(* Logix 5000 project; controller Google vendor 1 type 14 code 151 rev 31.11; software revision 31.00; part 3 of 5 *)
(* tags used below, declared in another part *)
   API_AcceptFromAgv : BOOL;
   API_ScanRequest : BOOL;
   API_ScanRequestFWDTimer : TIMER;
   API_SendToAgv : BOOL;
   API_SendToAgvTimer : TIMER;
   Elev_FWD_Delay : TIMER;
   Elev_REV_Delay : TIMER;
   Elev_Slow : BOOL;
   FaultResetDelay : TIMER;
   HMI_AutoMode : BOOL;
   HMI_LiftJogDown : BOOL;
   HMI_LiftJogUp : BOOL;
   HMI_PB_Reset : BOOL;
   Infeed_Active : BOOL;
   Infeed_Upstream_ProdCode : DINT;
   Infeed_Upstream_ProdName : STRING;
   Infeed_Zone1 : Zone_Data;
   Infeed_Zone1_2_ProdCode : DINT;
   Infeed_Zone1_2_ProdName : STRING;
   Infeed_Zone1_FWD : BOOL;
   Infeed_Zone1_PE : BOOL;
   Infeed_Zone1_ProdCode : DINT;
   Infeed_Zone1_ProdName : STRING;
   Infeed_Zone1_REV : BOOL;
   Infeed_Zone2 : Zone_Data;
   Infeed_Zone2_3_ProdCode : DINT;
   Infeed_Zone2_3_ProdName : STRING;
   Infeed_Zone2_FWD : BOOL;
   Infeed_Zone2_PE : BOOL;
   Infeed_Zone2_ProdCode : DINT;
   Infeed_Zone2_ProdName : STRING;
   Infeed_Zone2_REV : BOOL;
   Infeed_Zone3 : Zone_Data;
   Infeed_Zone3_4_ProdCode : DINT;
   Infeed_Zone3_4_ProdName : STRING;
   Infeed_Zone3_FWD : BOOL;
   Infeed_Zone3_PE : BOOL;
   Infeed_Zone3_ProdCode : DINT;
   Infeed_Zone3_ProdName : STRING;
   Infeed_Zone3_REV : BOOL;
   Infeed_Zone4 : Zone_Data;
   Infeed_Zone4_FWD : BOOL;
   Infeed_Zone4_PE : BOOL;
   Infeed_Zone4_ProdCode : DINT;
   Infeed_Zone4_ProdName : STRING;
   Infeed_Zone4_REV : BOOL;
   Infeed_Zone_Timeout : TIMER[8];
   L1_CearOutResetTimer : TIMER;
   L1_Clear_Out : BOOL;
   L1_Zone1_FWD : BOOL;
   L1_Zone1_PE : BOOL;
   L2_Outfeed : BOOL;
   L2_Single_Outfeed : BOOL;
   L2_Z1_Outfeed : BOOL;
   L2_Z2_Outfeed : BOOL;
   L2_Z3_Outfeed : BOOL;
   L2_Z4_Outfeed : BOOL;
   L2_Zone1 : Zone_Data;
   L2_Zone2 : Zone_Data;
   L2_Zone3 : Zone_Data;
   L3_Outfeed : BOOL;
   L3_Single_Outfeed : BOOL;
   L3_Z1_Outfeed : BOOL;
   L3_Z2_Outfeed : BOOL;
   L3_Z3_Outfeed : BOOL;
   L3_Z4_Outfeed : BOOL;
   L3_Zone1 : Zone_Data;
   L3_Zone2 : Zone_Data;
   L3_Zone3 : Zone_Data;
   L4_Outfeed : BOOL;
   L4_Single_Outfeed : BOOL;
   L4_Z1_Outfeed : BOOL;
   L4_Z2_Outfeed : BOOL;
   L4_Z3_Outfeed : BOOL;
   L4_Z4_Outfeed : BOOL;
   L4_Zone1 : Zone_Data;
   L4_Zone2 : Zone_Data;
   L4_Zone3 : Zone_Data;
   L5_Outfeed : BOOL;
   L5_Single_Outfeed : BOOL;
   L5_Z1_Outfeed : BOOL;
   L5_Z2_Outfeed : BOOL;
   L5_Z3_Outfeed : BOOL;
   L5_Z4_Outfeed : BOOL;
   L5_Zone1 : Zone_Data;
   L5_Zone2 : Zone_Data;
   L5_Zone3 : Zone_Data;
   Level_1_Empty : BOOL;
   Level_2_Empty : BOOL;
   Level_2_Full : BOOL;
   Level_3_Empty : BOOL;
   Level_3_Full : BOOL;
   Level_4_Empty : BOOL;
   Level_4_Full : BOOL;
   Level_5_Empty : BOOL;
   Level_5_Full : BOOL;
   Lift_Alarm : BOOL;
   Lift_Ascend : BOOL;
   Lift_Current_Level : DINT;
   Lift_Cycle_Counter : COUNTER;
   Lift_Descend : BOOL;
   Lift_FullSpeed : DINT;
   Lift_L1_Slow_Prox : BOOL;
   Lift_L1_Stop_Prox : BOOL;
   Lift_L2_Slow_Prox : BOOL;
   Lift_L2_Stop_Prox : BOOL;
   Lift_L3_Slow_Prox : BOOL;
   Lift_L3_Stop_Prox : BOOL;
   Lift_L4_Slow_Prox : BOOL;
   Lift_L4_Stop_Prox : BOOL;
   Lift_L5_Slow_Prox : BOOL;
   Lift_L5_Stop_Prox : BOOL;
   Lift_Required_Level : DINT;
   Lift_SlowSpeed : DINT;
   Lift_Zone : Lift_Zone_Data;
   LiftZone_FWD : BOOL;
   LiftZone_REV : BOOL;
   LiftZoneDownstream_ProdCode : DINT;
   LiftZoneUpstream_ProdName : STRING;
   Motion_Complete : BOOL;
   ONS : DINT[6];
   Outfeed_Active : BOOL;
   Outfeed_Automatic : BOOL;
   Outfeed_Batch : BOOL;
   Outfeed_Single : BOOL;
   Safety_Relay_Status : BOOL;
   Sort_Number : DINT;
   Sorting_Active : BOOL;
   Sorting_Inactive : BOOL;
   System : State;
   System_Mode_Change : BOOL;
   System_State : DINT;
(* MainProgram, continued *)

ROUTINE R04_Sorting   (* ladder *)
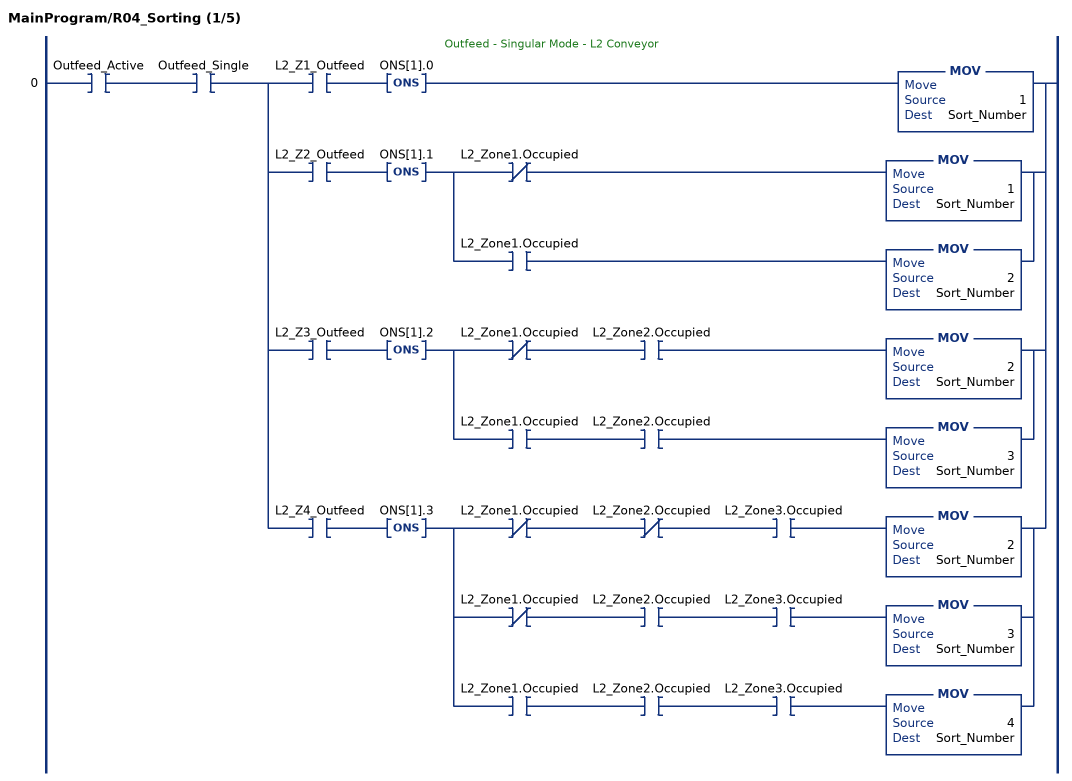
   // Outfeed - Singular Mode - L2 Conveyor
   0: XIC(Outfeed_Active)XIC(Outfeed_Single)[XIC(L2_Z1_Outfeed) ONS(ONS[1].0) MOV(1,Sort_Number) ,XIC(L2_Z2_Outfeed) ONS(ONS[1].1) [XIO(L2_Zone1.Occupied) MOV(1,Sort_Number) ,XIC(L2_Zone1.Occupied) MOV(2,Sort_Number) ] ,XIC(L2_Z3_Outfeed) ONS(ONS[1].2) [XIO(L2_Zone1.Occupied) XIC(L2_Zone2.Occupied) MOV(2,Sort_Number) ,XIC(L2_Zone1.Occupied) XIC(L2_Zone2.Occupied) MOV(3,Sort_Number) ] ,XIC(L2_Z4_Outfeed) ONS(ONS[1].3) [XIO(L2_Zone1.Occupied) XIO(L2_Zone2.Occupied) XIC(L2_Zone3.Occupied) MOV(2,Sort_Number) ,XIO(L2_Zone1.Occupied) XIC(L2_Zone2.Occupied) XIC(L2_Zone3.Occupied) MOV(3,Sort_Number) ,XIC(L2_Zone1.Occupied) XIC(L2_Zone2.Occupied) XIC(L2_Zone3.Occupied) MOV(4,Sort_Number) ] ];
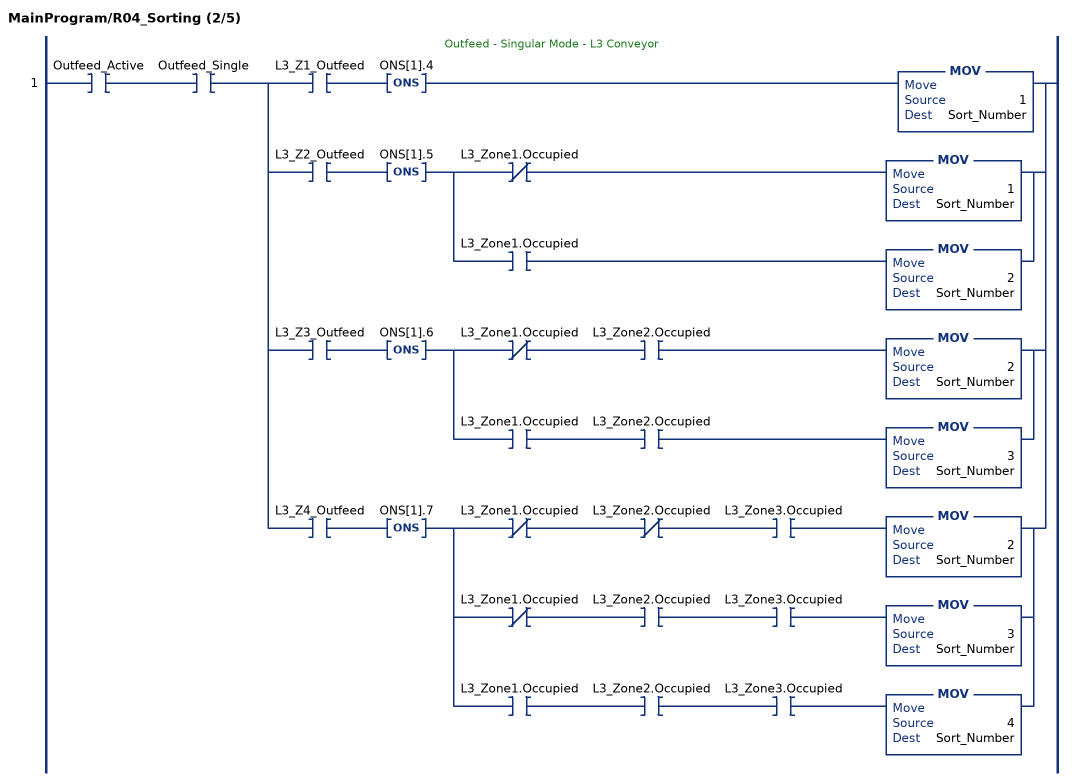
   // Outfeed - Singular Mode - L3 Conveyor
   1: XIC(Outfeed_Active)XIC(Outfeed_Single)[XIC(L3_Z1_Outfeed) ONS(ONS[1].4) MOV(1,Sort_Number) ,XIC(L3_Z2_Outfeed) ONS(ONS[1].5) [XIO(L3_Zone1.Occupied) MOV(1,Sort_Number) ,XIC(L3_Zone1.Occupied) MOV(2,Sort_Number) ] ,XIC(L3_Z3_Outfeed) ONS(ONS[1].6) [XIO(L3_Zone1.Occupied) XIC(L3_Zone2.Occupied) MOV(2,Sort_Number) ,XIC(L3_Zone1.Occupied) XIC(L3_Zone2.Occupied) MOV(3,Sort_Number) ] ,XIC(L3_Z4_Outfeed) ONS(ONS[1].7) [XIO(L3_Zone1.Occupied) XIO(L3_Zone2.Occupied) XIC(L3_Zone3.Occupied) MOV(2,Sort_Number) ,XIO(L3_Zone1.Occupied) XIC(L3_Zone2.Occupied) XIC(L3_Zone3.Occupied) MOV(3,Sort_Number) ,XIC(L3_Zone1.Occupied) XIC(L3_Zone2.Occupied) XIC(L3_Zone3.Occupied) MOV(4,Sort_Number) ] ];
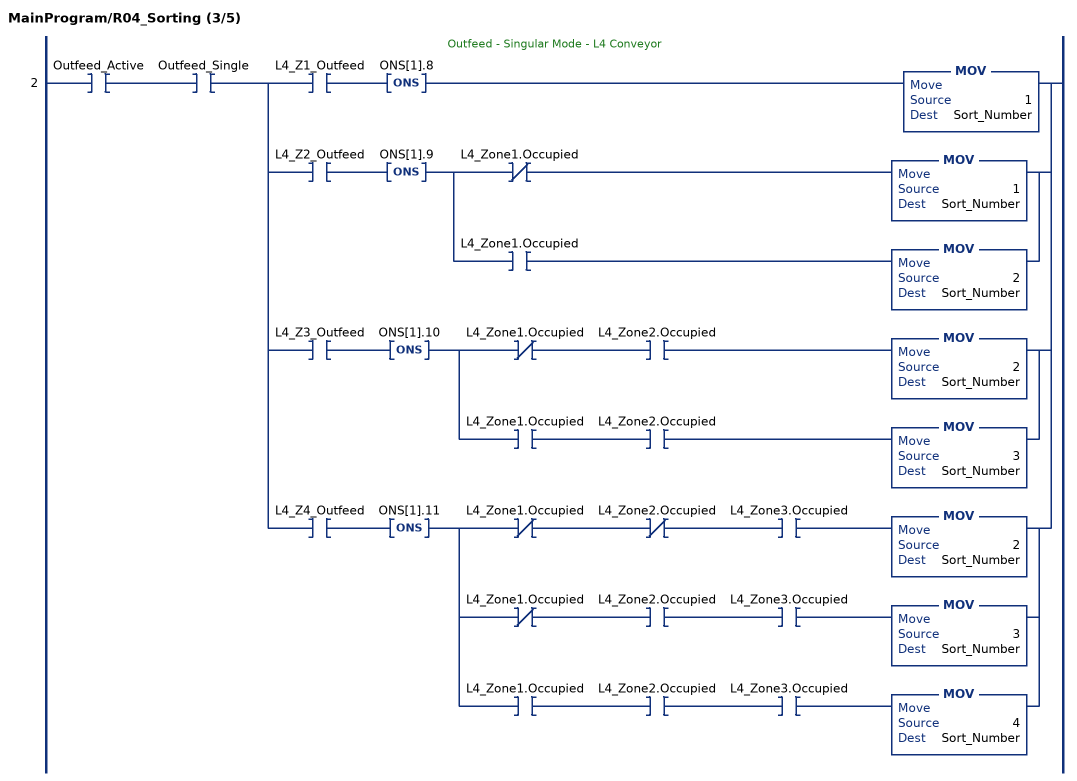
   // Outfeed - Singular Mode - L4 Conveyor
   2: XIC(Outfeed_Active)XIC(Outfeed_Single)[XIC(L4_Z1_Outfeed) ONS(ONS[1].8) MOV(1,Sort_Number) ,XIC(L4_Z2_Outfeed) ONS(ONS[1].9) [XIO(L4_Zone1.Occupied) MOV(1,Sort_Number) ,XIC(L4_Zone1.Occupied) MOV(2,Sort_Number) ] ,XIC(L4_Z3_Outfeed) ONS(ONS[1].10) [XIO(L4_Zone1.Occupied) XIC(L4_Zone2.Occupied) MOV(2,Sort_Number) ,XIC(L4_Zone1.Occupied) XIC(L4_Zone2.Occupied) MOV(3,Sort_Number) ] ,XIC(L4_Z4_Outfeed) ONS(ONS[1].11) [XIO(L4_Zone1.Occupied) XIO(L4_Zone2.Occupied) XIC(L4_Zone3.Occupied) MOV(2,Sort_Number) ,XIO(L4_Zone1.Occupied) XIC(L4_Zone2.Occupied) XIC(L4_Zone3.Occupied) MOV(3,Sort_Number) ,XIC(L4_Zone1.Occupied) XIC(L4_Zone2.Occupied) XIC(L4_Zone3.Occupied) MOV(4,Sort_Number) ] ];
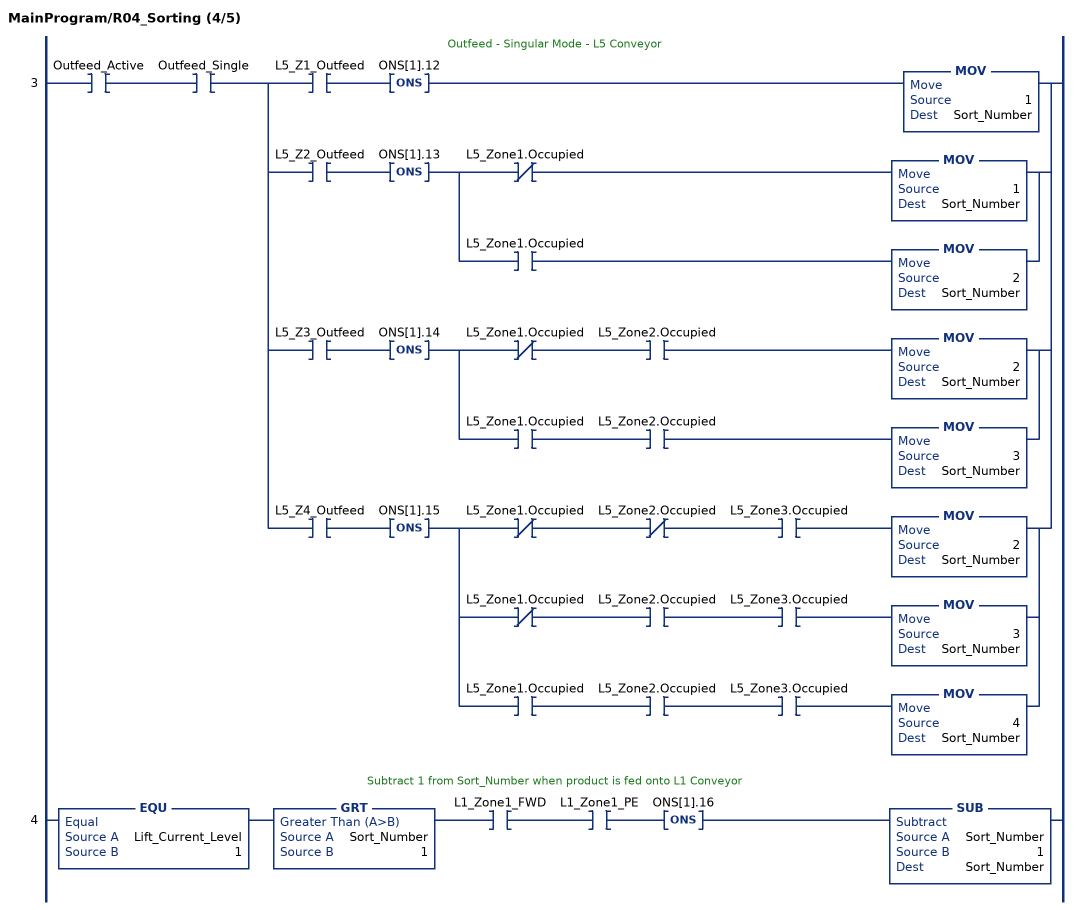
   // Outfeed - Singular Mode - L5 Conveyor
   3: XIC(Outfeed_Active)XIC(Outfeed_Single)[XIC(L5_Z1_Outfeed) ONS(ONS[1].12) MOV(1,Sort_Number) ,XIC(L5_Z2_Outfeed) ONS(ONS[1].13) [XIO(L5_Zone1.Occupied) MOV(1,Sort_Number) ,XIC(L5_Zone1.Occupied) MOV(2,Sort_Number) ] ,XIC(L5_Z3_Outfeed) ONS(ONS[1].14) [XIO(L5_Zone1.Occupied) XIC(L5_Zone2.Occupied) MOV(2,Sort_Number) ,XIC(L5_Zone1.Occupied) XIC(L5_Zone2.Occupied) MOV(3,Sort_Number) ] ,XIC(L5_Z4_Outfeed) ONS(ONS[1].15) [XIO(L5_Zone1.Occupied) XIO(L5_Zone2.Occupied) XIC(L5_Zone3.Occupied) MOV(2,Sort_Number) ,XIO(L5_Zone1.Occupied) XIC(L5_Zone2.Occupied) XIC(L5_Zone3.Occupied) MOV(3,Sort_Number) ,XIC(L5_Zone1.Occupied) XIC(L5_Zone2.Occupied) XIC(L5_Zone3.Occupied) MOV(4,Sort_Number) ] ];
   // Subtract 1 from Sort_Number when product is fed onto L1 Conveyor
   4: EQU(Lift_Current_Level,1)GRT(Sort_Number,1)XIC(L1_Zone1_FWD)XIC(L1_Zone1_PE)ONS(ONS[1].16)SUB(Sort_Number,1,Sort_Number);
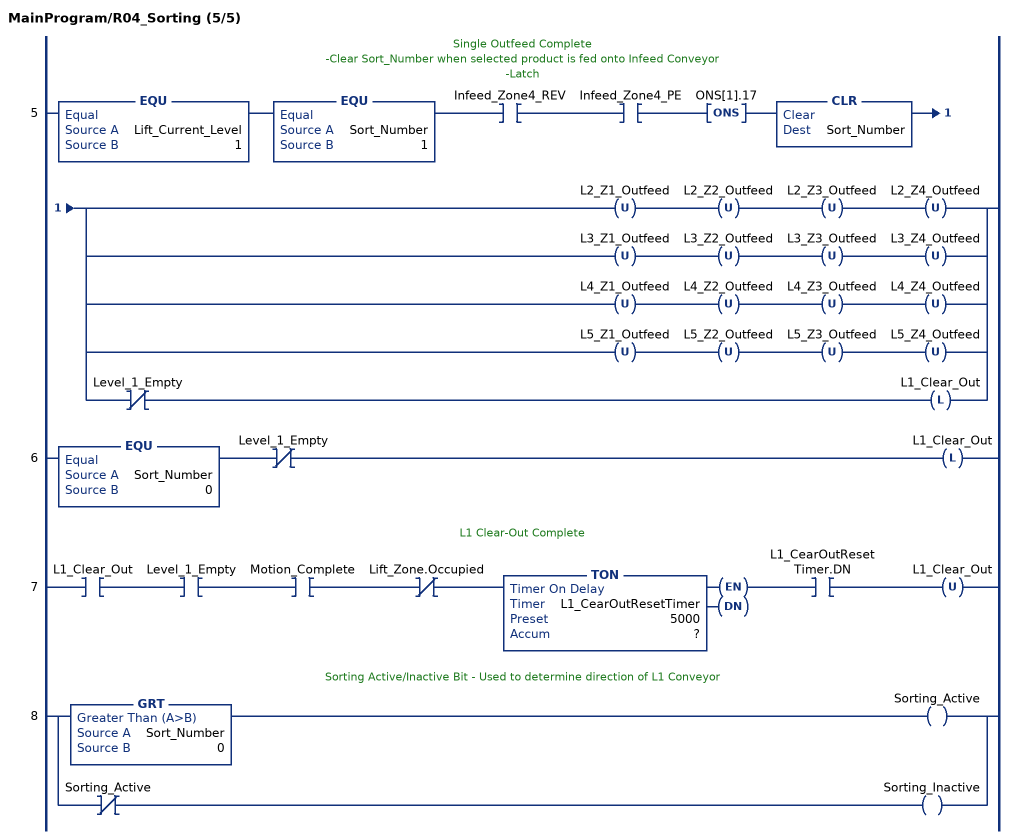
   // Single Outfeed Complete
   // -Clear Sort_Number when selected product is fed onto Infeed Conveyor
   // -Latch
   5: EQU(Lift_Current_Level,1)EQU(Sort_Number,1)XIC(Infeed_Zone4_REV)XIC(Infeed_Zone4_PE)ONS(ONS[1].17)CLR(Sort_Number)[OTU(L2_Z1_Outfeed) OTU(L2_Z2_Outfeed) OTU(L2_Z3_Outfeed) OTU(L2_Z4_Outfeed) ,OTU(L3_Z1_Outfeed) OTU(L3_Z2_Outfeed) OTU(L3_Z3_Outfeed) OTU(L3_Z4_Outfeed) ,OTU(L4_Z1_Outfeed) OTU(L4_Z2_Outfeed) OTU(L4_Z3_Outfeed) OTU(L4_Z4_Outfeed) ,OTU(L5_Z1_Outfeed) OTU(L5_Z2_Outfeed) OTU(L5_Z3_Outfeed) OTU(L5_Z4_Outfeed) ,XIO(Level_1_Empty) OTL(L1_Clear_Out) ];
   6: EQU(Sort_Number,0)XIO(Level_1_Empty)OTL(L1_Clear_Out);
   // L1 Clear-Out Complete
   7: XIC(L1_Clear_Out)XIC(Level_1_Empty)XIC(Motion_Complete)XIO(Lift_Zone.Occupied)TON(L1_CearOutResetTimer,?,?)XIC(L1_CearOutResetTimer.DN)OTU(L1_Clear_Out);
   // Sorting Active/Inactive Bit - Used to determine direction of L1 Conveyor
   8: [GRT(Sort_Number,0) OTE(Sorting_Active) ,XIO(Sorting_Active) OTE(Sorting_Inactive) ];
END_ROUTINE

ROUTINE R05_Lift_Level_Selection   (* ladder *)
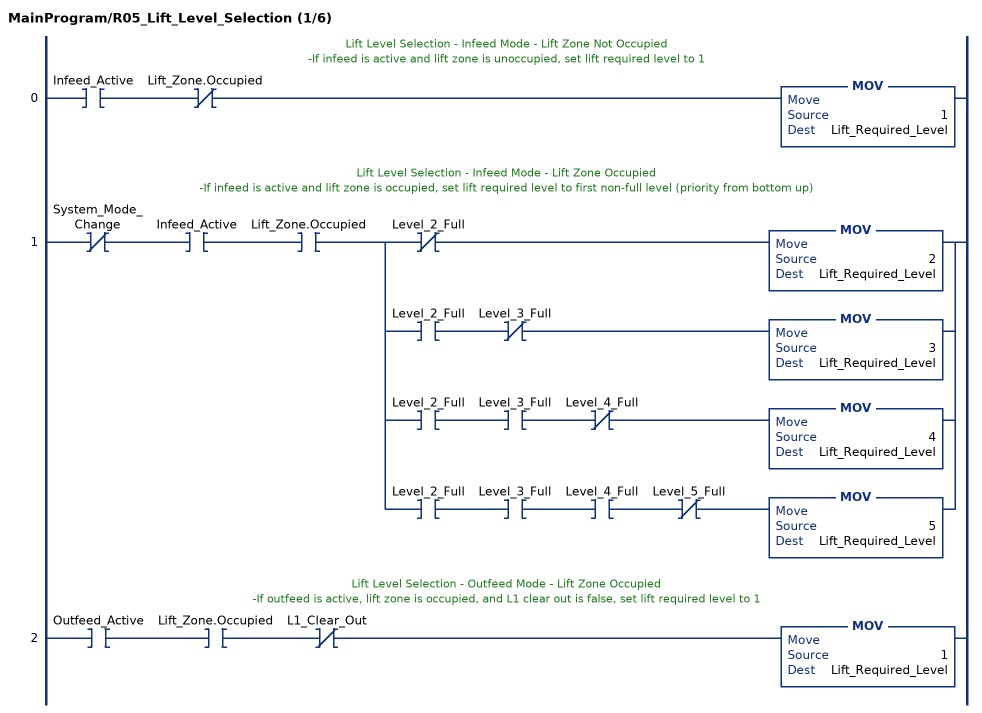
   // Lift Level Selection - Infeed Mode - Lift Zone Not Occupied
   // -If infeed is active and lift zone is unoccupied, set lift required level to 1
   0: XIC(Infeed_Active)XIO(Lift_Zone.Occupied)MOV(1,Lift_Required_Level);
   // Lift Level Selection - Infeed Mode - Lift Zone Occupied
   // -If infeed is active and lift zone is occupied, set lift required level to first non-full level (priority from bottom up)
   1: XIO(System_Mode_Change)XIC(Infeed_Active)XIC(Lift_Zone.Occupied)[XIO(Level_2_Full) MOV(2,Lift_Required_Level) ,XIC(Level_2_Full) XIO(Level_3_Full) MOV(3,Lift_Required_Level) ,XIC(Level_2_Full) XIC(Level_3_Full) XIO(Level_4_Full) MOV(4,Lift_Required_Level) ,XIC(Level_2_Full) XIC(Level_3_Full) XIC(Level_4_Full) XIO(Level_5_Full) MOV(5,Lift_Required_Level) ];
   // Lift Level Selection - Outfeed Mode - Lift Zone Occupied
   // -If outfeed is active, lift zone is occupied, and L1 clear out is false, set lift required level to 1
   2: XIC(Outfeed_Active)XIC(Lift_Zone.Occupied)XIO(L1_Clear_Out)MOV(1,Lift_Required_Level);
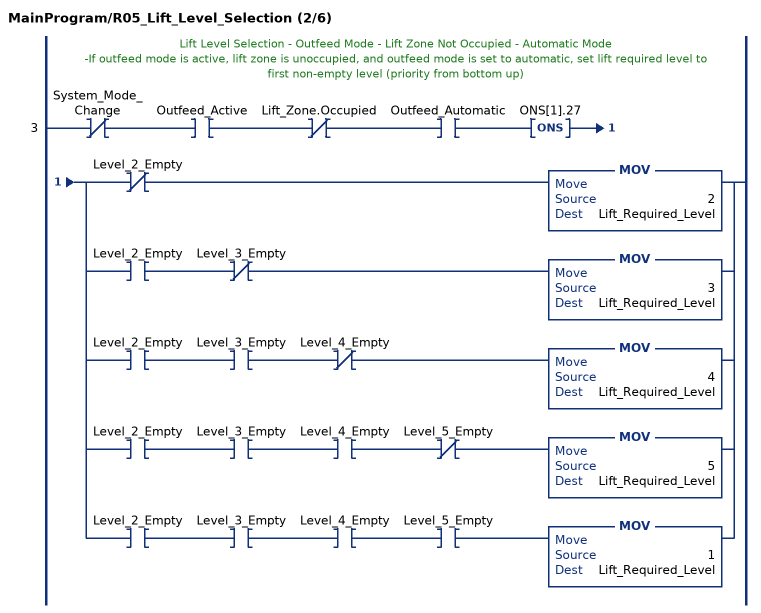
   // Lift Level Selection - Outfeed Mode - Lift Zone Not Occupied - Automatic Mode
   // -If outfeed mode is active, lift zone is unoccupied, and outfeed mode is set to automatic, set lift required level to first non-empty level (priority from bottom up)
   3: XIO(System_Mode_Change)XIC(Outfeed_Active)XIO(Lift_Zone.Occupied)XIC(Outfeed_Automatic)ONS(ONS[1].27)[XIO(Level_2_Empty) MOV(2,Lift_Required_Level) ,XIC(Level_2_Empty) XIO(Level_3_Empty) MOV(3,Lift_Required_Level) ,XIC(Level_2_Empty) XIC(Level_3_Empty) XIO(Level_4_Empty) MOV(4,Lift_Required_Level) ,XIC(Level_2_Empty) XIC(Level_3_Empty) XIC(Level_4_Empty) XIO(Level_5_Empty) MOV(5,Lift_Required_Level) ,XIC(Level_2_Empty) XIC(Level_3_Empty) XIC(Level_4_Empty) XIC(Level_5_Empty) MOV(1,Lift_Required_Level) ];
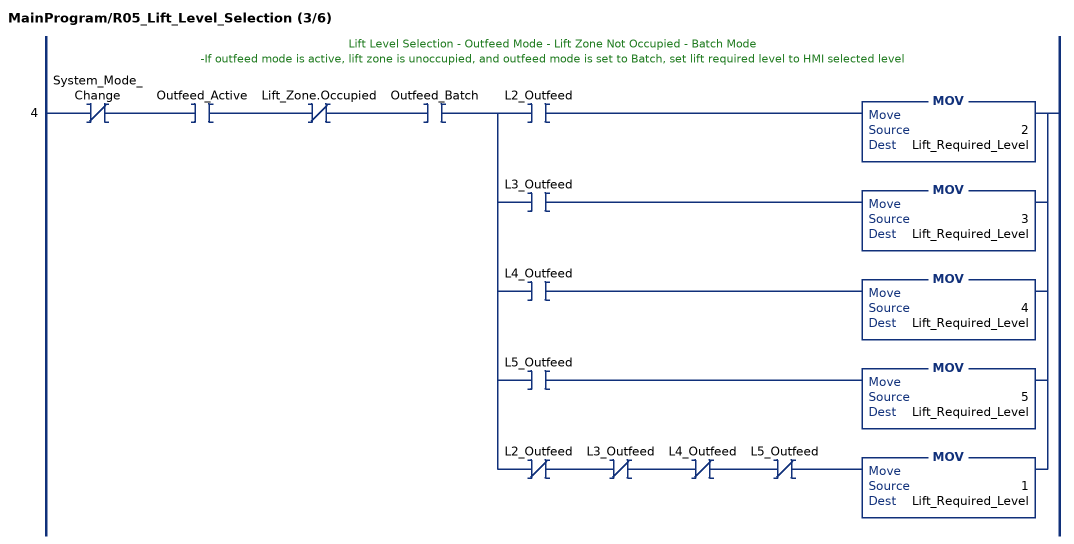
   // Lift Level Selection - Outfeed Mode - Lift Zone Not Occupied - Batch Mode
   // -If outfeed mode is active, lift zone is unoccupied, and outfeed mode is set to Batch, set lift required level to HMI selected level
   4: XIO(System_Mode_Change)XIC(Outfeed_Active)XIO(Lift_Zone.Occupied)XIC(Outfeed_Batch)[XIC(L2_Outfeed) MOV(2,Lift_Required_Level) ,XIC(L3_Outfeed) MOV(3,Lift_Required_Level) ,XIC(L4_Outfeed) MOV(4,Lift_Required_Level) ,XIC(L5_Outfeed) MOV(5,Lift_Required_Level) ,XIO(L2_Outfeed) XIO(L3_Outfeed) XIO(L4_Outfeed) XIO(L5_Outfeed) MOV(1,Lift_Required_Level) ];
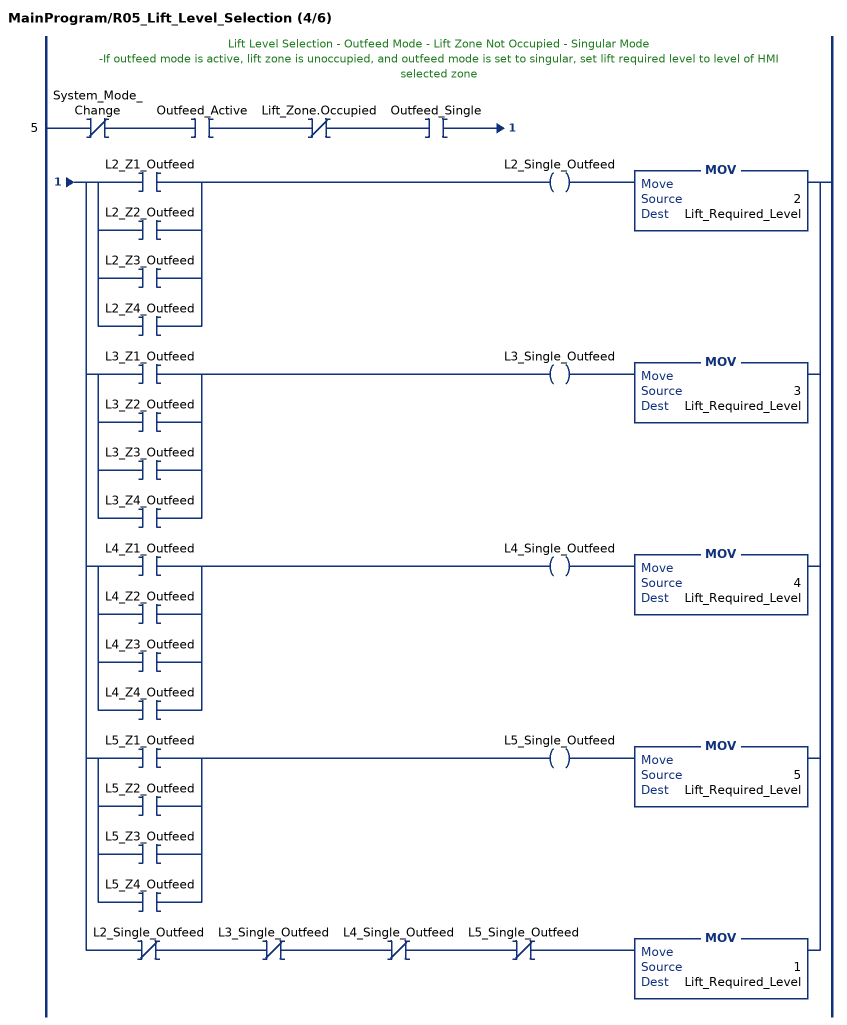
   // Lift Level Selection - Outfeed Mode - Lift Zone Not Occupied - Singular Mode
   // -If outfeed mode is active, lift zone is unoccupied, and outfeed mode is set to singular, set lift required level to level of HMI selected zone
   5: XIO(System_Mode_Change)XIC(Outfeed_Active)XIO(Lift_Zone.Occupied)XIC(Outfeed_Single)[[XIC(L2_Z1_Outfeed) ,XIC(L2_Z2_Outfeed) ,XIC(L2_Z3_Outfeed) ,XIC(L2_Z4_Outfeed) ] OTE(L2_Single_Outfeed) MOV(2,Lift_Required_Level) ,[XIC(L3_Z1_Outfeed) ,XIC(L3_Z2_Outfeed) ,XIC(L3_Z3_Outfeed) ,XIC(L3_Z4_Outfeed) ] OTE(L3_Single_Outfeed) MOV(3,Lift_Required_Level) ,[XIC(L4_Z1_Outfeed) ,XIC(L4_Z2_Outfeed) ,XIC(L4_Z3_Outfeed) ,XIC(L4_Z4_Outfeed) ] OTE(L4_Single_Outfeed) MOV(4,Lift_Required_Level) ,[XIC(L5_Z1_Outfeed) ,XIC(L5_Z2_Outfeed) ,XIC(L5_Z3_Outfeed) ,XIC(L5_Z4_Outfeed) ] OTE(L5_Single_Outfeed) MOV(5,Lift_Required_Level) ,XIO(L2_Single_Outfeed) XIO(L3_Single_Outfeed) XIO(L4_Single_Outfeed) XIO(L5_Single_Outfeed) MOV(1,Lift_Required_Level) ];
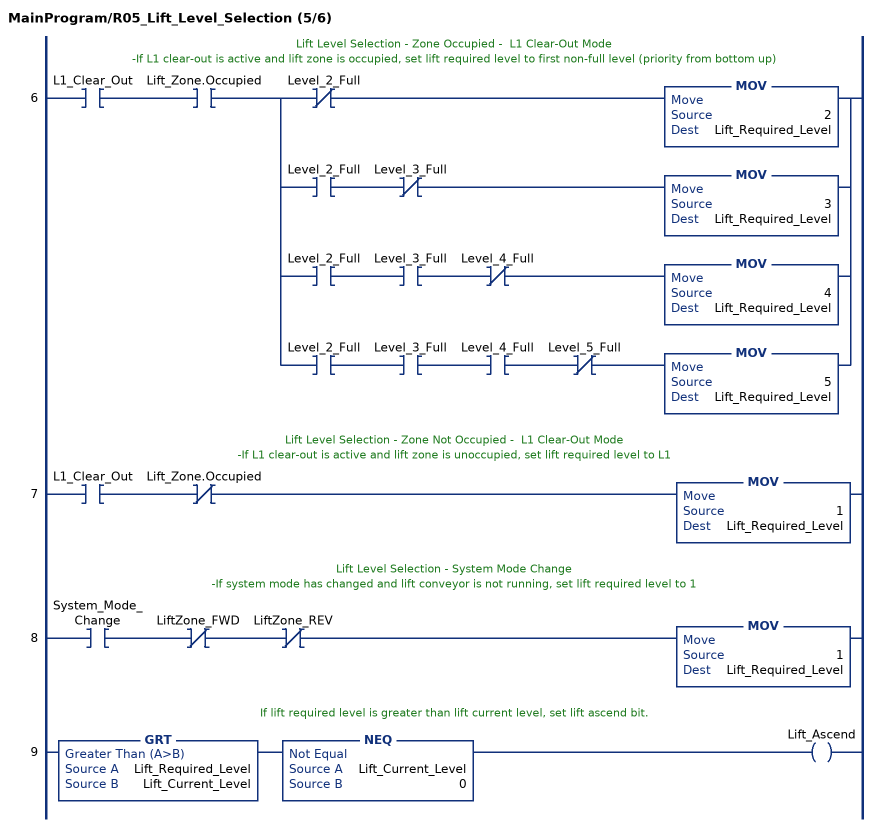
   // Lift Level Selection - Zone Occupied -  L1 Clear-Out Mode
   // -If L1 clear-out is active and lift zone is occupied, set lift required level to first non-full level (priority from bottom up)
   6: XIC(L1_Clear_Out)XIC(Lift_Zone.Occupied)[XIO(Level_2_Full) MOV(2,Lift_Required_Level) ,XIC(Level_2_Full) XIO(Level_3_Full) MOV(3,Lift_Required_Level) ,XIC(Level_2_Full) XIC(Level_3_Full) XIO(Level_4_Full) MOV(4,Lift_Required_Level) ,XIC(Level_2_Full) XIC(Level_3_Full) XIC(Level_4_Full) XIO(Level_5_Full) MOV(5,Lift_Required_Level) ];
   // Lift Level Selection - Zone Not Occupied -  L1 Clear-Out Mode
   // -If L1 clear-out is active and lift zone is unoccupied, set lift required level to L1
   7: XIC(L1_Clear_Out)XIO(Lift_Zone.Occupied)MOV(1,Lift_Required_Level);
   // Lift Level Selection - System Mode Change
   // -If system mode has changed and lift conveyor is not running, set lift required level to 1
   8: XIC(System_Mode_Change)XIO(LiftZone_FWD)XIO(LiftZone_REV)MOV(1,Lift_Required_Level);
   // If lift required level is greater than lift current level, set lift ascend bit.
   9: GRT(Lift_Required_Level,Lift_Current_Level)NEQ(Lift_Current_Level,0)OTE(Lift_Ascend);
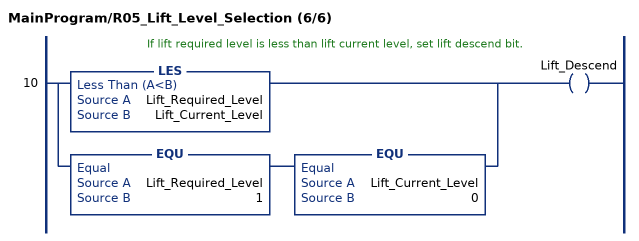
   // If lift required level is less than lift current level, set lift descend bit.
   10: [LES(Lift_Required_Level,Lift_Current_Level) ,EQU(Lift_Required_Level,1) EQU(Lift_Current_Level,0) ]OTE(Lift_Descend);
END_ROUTINE

ROUTINE R06_Lift_Operation   (* ladder *)
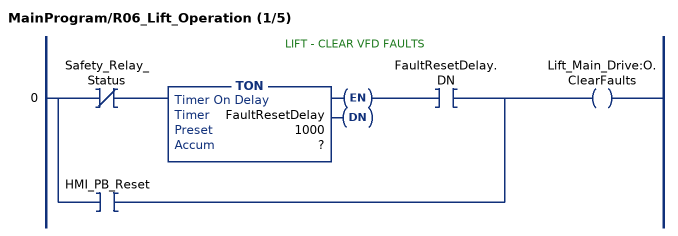
   // LIFT - CLEAR VFD FAULTS
   0: [XIO(Safety_Relay_Status) TON(FaultResetDelay,?,?) XIC(FaultResetDelay.DN) ,XIC(HMI_PB_Reset) ]OTE(Lift_Main_Drive:O.ClearFaults);
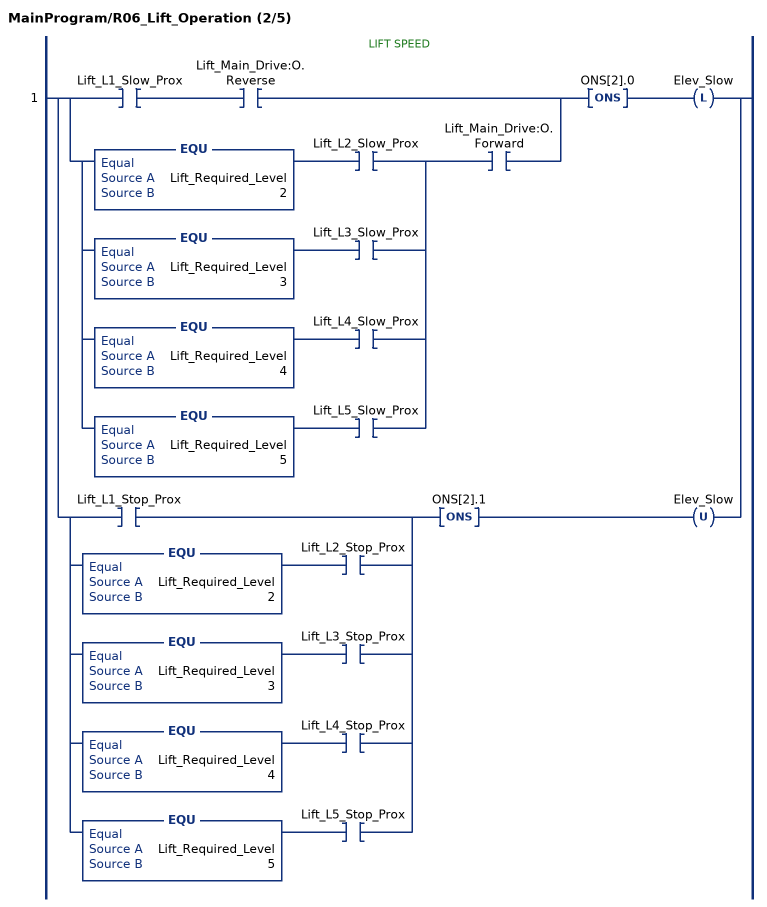
   // LIFT SPEED
   1: [[XIC(Lift_L1_Slow_Prox) XIC(Lift_Main_Drive:O.Reverse) ,[EQU(Lift_Required_Level,2) XIC(Lift_L2_Slow_Prox) ,EQU(Lift_Required_Level,3) XIC(Lift_L3_Slow_Prox) ,EQU(Lift_Required_Level,4) XIC(Lift_L4_Slow_Prox) ,EQU(Lift_Required_Level,5) XIC(Lift_L5_Slow_Prox) ] XIC(Lift_Main_Drive:O.Forward) ] ONS(ONS[2].0) OTL(Elev_Slow) ,[XIC(Lift_L1_Stop_Prox) ,EQU(Lift_Required_Level,2) XIC(Lift_L2_Stop_Prox) ,EQU(Lift_Required_Level,3) XIC(Lift_L3_Stop_Prox) ,EQU(Lift_Required_Level,4) XIC(Lift_L4_Stop_Prox) ,EQU(Lift_Required_Level,5) XIC(Lift_L5_Stop_Prox) ] ONS(ONS[2].1) OTU(Elev_Slow) ];
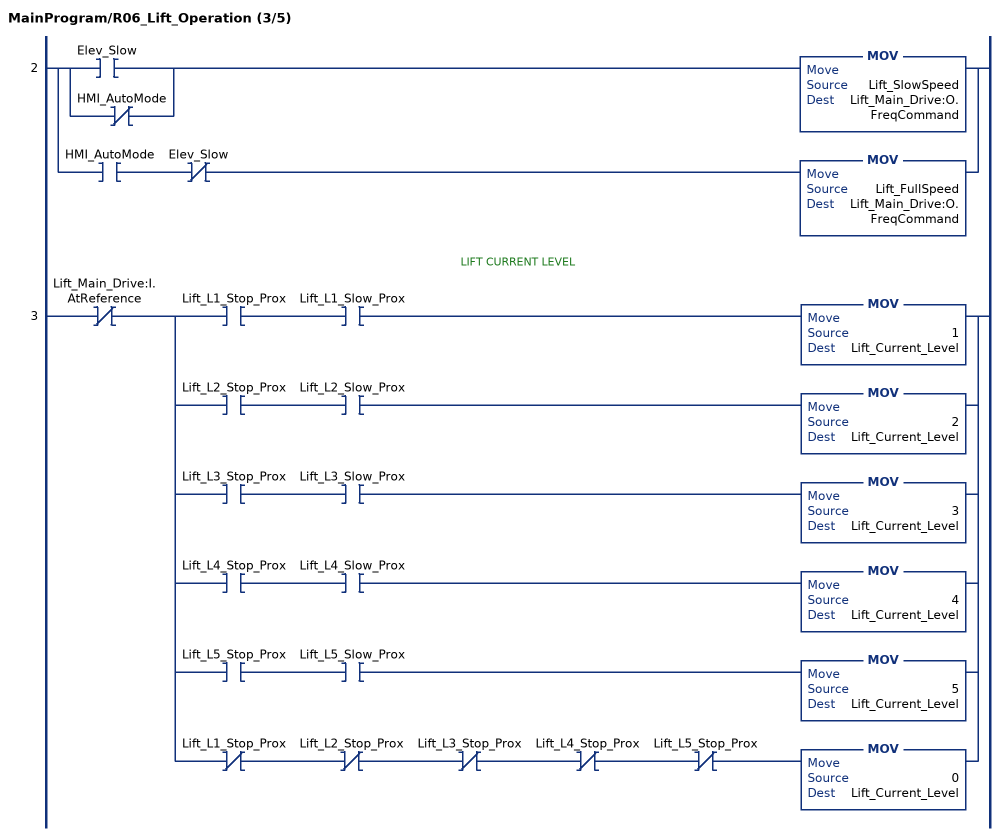
   2: [[XIC(Elev_Slow) ,XIO(HMI_AutoMode) ] MOV(Lift_SlowSpeed,Lift_Main_Drive:O.FreqCommand) ,XIC(HMI_AutoMode) XIO(Elev_Slow) MOV(Lift_FullSpeed,Lift_Main_Drive:O.FreqCommand) ];
   // LIFT CURRENT LEVEL
   3: XIO(Lift_Main_Drive:I.AtReference)[XIC(Lift_L1_Stop_Prox) XIC(Lift_L1_Slow_Prox) MOV(1,Lift_Current_Level) ,XIC(Lift_L2_Stop_Prox) XIC(Lift_L2_Slow_Prox) MOV(2,Lift_Current_Level) ,XIC(Lift_L3_Stop_Prox) XIC(Lift_L3_Slow_Prox) MOV(3,Lift_Current_Level) ,XIC(Lift_L4_Stop_Prox) XIC(Lift_L4_Slow_Prox) MOV(4,Lift_Current_Level) ,XIC(Lift_L5_Stop_Prox) XIC(Lift_L5_Slow_Prox) MOV(5,Lift_Current_Level) ,XIO(Lift_L1_Stop_Prox) XIO(Lift_L2_Stop_Prox) XIO(Lift_L3_Stop_Prox) XIO(Lift_L4_Stop_Prox) XIO(Lift_L5_Stop_Prox) MOV(0,Lift_Current_Level) ];
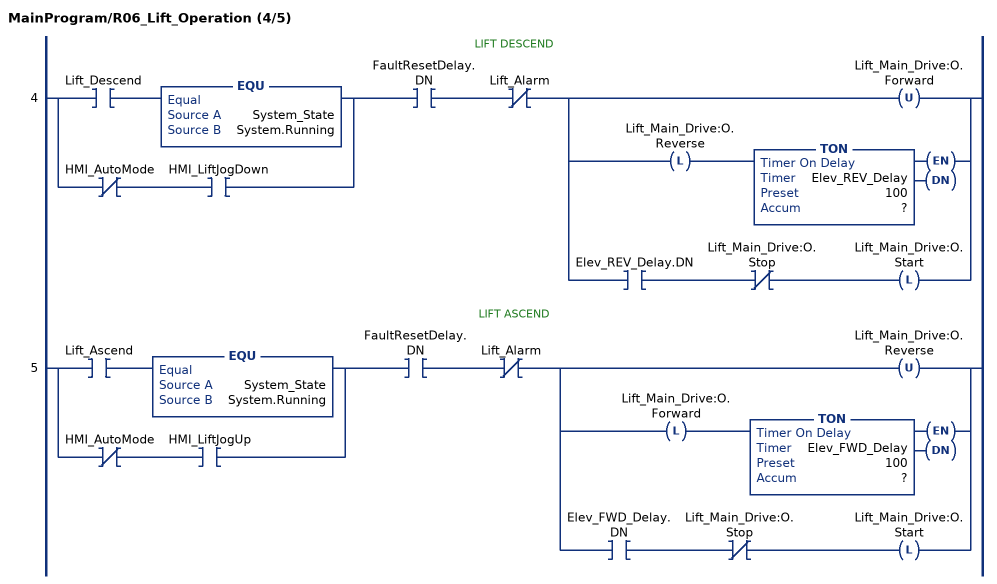
   // LIFT DESCEND
   4: [XIC(Lift_Descend) EQU(System_State,System.Running) ,XIO(HMI_AutoMode) XIC(HMI_LiftJogDown) ]XIC(FaultResetDelay.DN)XIO(Lift_Alarm)[OTU(Lift_Main_Drive:O.Forward) ,OTL(Lift_Main_Drive:O.Reverse) TON(Elev_REV_Delay,?,?) ,XIC(Elev_REV_Delay.DN) XIO(Lift_Main_Drive:O.Stop) OTL(Lift_Main_Drive:O.Start) ];
   // LIFT ASCEND
   5: [XIC(Lift_Ascend) EQU(System_State,System.Running) ,XIO(HMI_AutoMode) XIC(HMI_LiftJogUp) ]XIC(FaultResetDelay.DN)XIO(Lift_Alarm)[OTU(Lift_Main_Drive:O.Reverse) ,OTL(Lift_Main_Drive:O.Forward) TON(Elev_FWD_Delay,?,?) ,XIC(Elev_FWD_Delay.DN) XIO(Lift_Main_Drive:O.Stop) OTL(Lift_Main_Drive:O.Start) ];
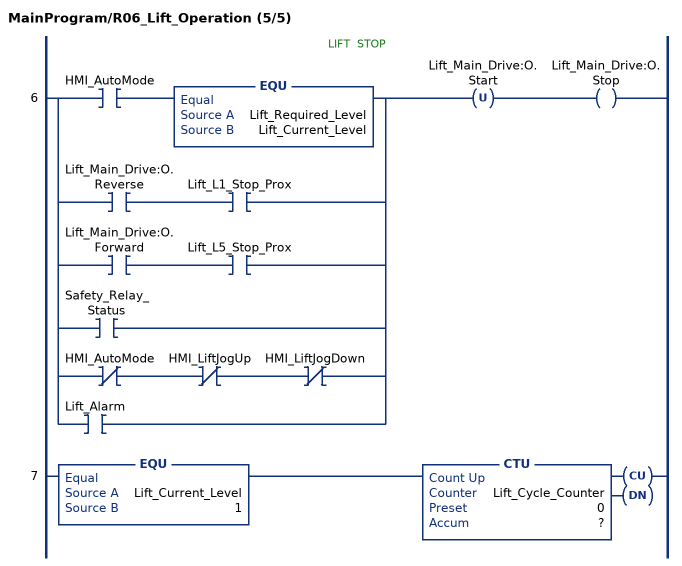
   // LIFT  STOP
   6: [XIC(HMI_AutoMode) EQU(Lift_Required_Level,Lift_Current_Level) ,XIC(Lift_Main_Drive:O.Reverse) XIC(Lift_L1_Stop_Prox) ,XIC(Lift_Main_Drive:O.Forward) XIC(Lift_L5_Stop_Prox) ,XIC(Safety_Relay_Status) ,XIO(HMI_AutoMode) XIO(HMI_LiftJogUp) XIO(HMI_LiftJogDown) ,XIC(Lift_Alarm) ]OTU(Lift_Main_Drive:O.Start)OTE(Lift_Main_Drive:O.Stop);
   7: EQU(Lift_Current_Level,1)CTU(Lift_Cycle_Counter,?,?);
END_ROUTINE

ROUTINE R07_Infeed_Conveyor   (* ladder *)
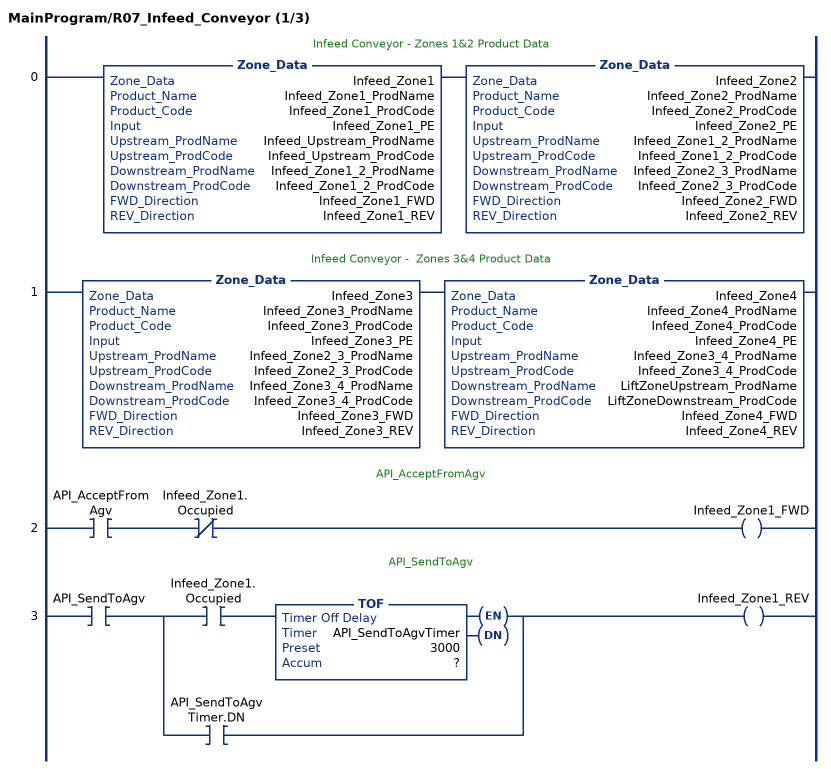
   // Infeed Conveyor - Zones 1&2 Product Data
   0: Zone_Data(Infeed_Zone1,Infeed_Zone1_ProdName,Infeed_Zone1_ProdCode,Infeed_Zone1_PE,Infeed_Upstream_ProdName,Infeed_Upstream_ProdCode,Infeed_Zone1_2_ProdName,Infeed_Zone1_2_ProdCode,Infeed_Zone1_FWD,Infeed_Zone1_REV)Zone_Data(Infeed_Zone2,Infeed_Zone2_ProdName,Infeed_Zone2_ProdCode,Infeed_Zone2_PE,Infeed_Zone1_2_ProdName,Infeed_Zone1_2_ProdCode,Infeed_Zone2_3_ProdName,Infeed_Zone2_3_ProdCode,Infeed_Zone2_FWD,Infeed_Zone2_REV);
   // Infeed Conveyor -  Zones 3&4 Product Data
   1: Zone_Data(Infeed_Zone3,Infeed_Zone3_ProdName,Infeed_Zone3_ProdCode,Infeed_Zone3_PE,Infeed_Zone2_3_ProdName,Infeed_Zone2_3_ProdCode,Infeed_Zone3_4_ProdName,Infeed_Zone3_4_ProdCode,Infeed_Zone3_FWD,Infeed_Zone3_REV)Zone_Data(Infeed_Zone4,Infeed_Zone4_ProdName,Infeed_Zone4_ProdCode,Infeed_Zone4_PE,Infeed_Zone3_4_ProdName,Infeed_Zone3_4_ProdCode,LiftZoneUpstream_ProdName,LiftZoneDownstream_ProdCode,Infeed_Zone4_FWD,Infeed_Zone4_REV);
   // API_AcceptFromAgv
   2: XIC(API_AcceptFromAgv)XIO(Infeed_Zone1.Occupied)OTE(Infeed_Zone1_FWD);
   // API_SendToAgv
   3: XIC(API_SendToAgv)[XIC(Infeed_Zone1.Occupied) TOF(API_SendToAgvTimer,?,?) ,XIC(API_SendToAgvTimer.DN) ]OTE(Infeed_Zone1_REV);
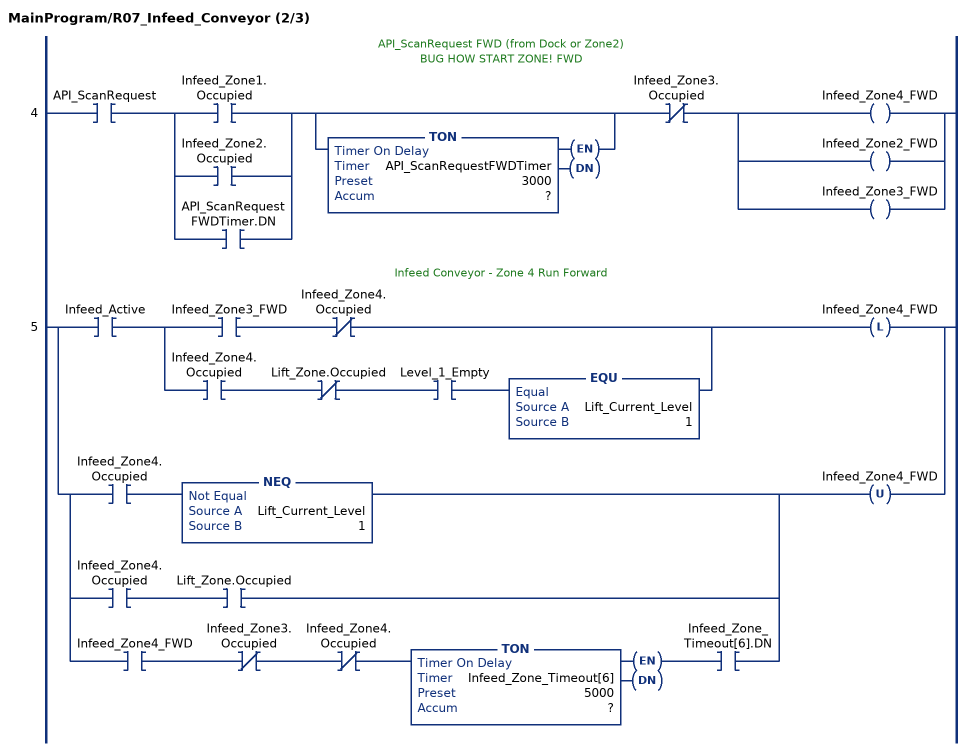
   // API_ScanRequest FWD (from Dock or Zone2)
   // BUG HOW START ZONE! FWD
   4: XIC(API_ScanRequest)[XIC(Infeed_Zone1.Occupied) ,XIC(Infeed_Zone2.Occupied) ,XIC(API_ScanRequestFWDTimer.DN) ][,TON(API_ScanRequestFWDTimer,?,?) ]XIO(Infeed_Zone3.Occupied)[OTE(Infeed_Zone4_FWD) ,OTE(Infeed_Zone2_FWD) ,OTE(Infeed_Zone3_FWD) ];
   // Infeed Conveyor - Zone 4 Run Forward
   5: [XIC(Infeed_Active) [XIC(Infeed_Zone3_FWD) XIO(Infeed_Zone4.Occupied) ,XIC(Infeed_Zone4.Occupied) XIO(Lift_Zone.Occupied) XIC(Level_1_Empty) EQU(Lift_Current_Level,1) ] OTL(Infeed_Zone4_FWD) ,[XIC(Infeed_Zone4.Occupied) NEQ(Lift_Current_Level,1) ,XIC(Infeed_Zone4.Occupied) XIC(Lift_Zone.Occupied) ,XIC(Infeed_Zone4_FWD) XIO(Infeed_Zone3.Occupied) XIO(Infeed_Zone4.Occupied) TON(Infeed_Zone_Timeout[6],?,?) XIC(Infeed_Zone_Timeout[6].DN) ] OTU(Infeed_Zone4_FWD) ];
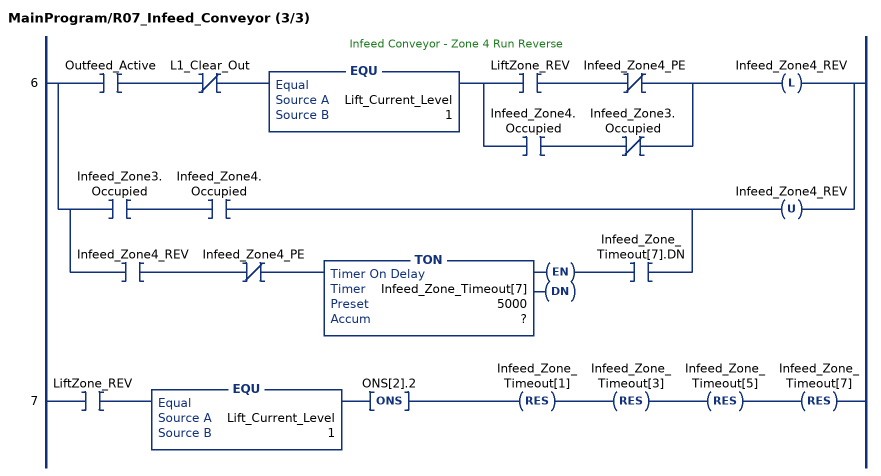
   // Infeed Conveyor - Zone 4 Run Reverse
   6: [XIC(Outfeed_Active) XIO(L1_Clear_Out) EQU(Lift_Current_Level,1) [XIC(LiftZone_REV) XIO(Infeed_Zone4_PE) ,XIC(Infeed_Zone4.Occupied) XIO(Infeed_Zone3.Occupied) ] OTL(Infeed_Zone4_REV) ,[XIC(Infeed_Zone3.Occupied) XIC(Infeed_Zone4.Occupied) ,XIC(Infeed_Zone4_REV) XIO(Infeed_Zone4_PE) TON(Infeed_Zone_Timeout[7],?,?) XIC(Infeed_Zone_Timeout[7].DN) ] OTU(Infeed_Zone4_REV) ];
   7: XIC(LiftZone_REV)EQU(Lift_Current_Level,1)ONS(ONS[2].2)RES(Infeed_Zone_Timeout[1])RES(Infeed_Zone_Timeout[3])RES(Infeed_Zone_Timeout[5])RES(Infeed_Zone_Timeout[7]);
END_ROUTINE
